// TIA Portal V18 export
DATA_BLOCK "DLsAI"   // DB51021
{ S7_Optimized_Access := 'FALSE' }
VERSION : 0.1
// stored: AutoNumber false, DBAccessibleFromOPCUA true, IsOnlyStoredInLoadMemory false, IsWriteProtectedInAS false
   VAR
      AI : "UDT_DLsAI";
   END_VAR
BEGIN
   AI.rDayTankLevel[1] := 0.0;
END_DATA_BLOCK
